(* CODESYS project Hylife_Repository

Project tree, tasks and I/O mapping:
  libraries: ; CXA_ModbusTCP, 1.8.0.3 (Bosch Rexroth AG)
  program PLC_PRG [ST]
*)

// PLC_PRG
PROGRAM PLC_PRG
VAR
	fbHandle_MB_CAN: FB_Handle_MB_CAN;
	//extra functie
	//Deze comment is toegevoegd vanuit een andere brench
	// test voor remote 2
	// test vor remote 
END_VAR

fbHandle_MB_CAN(I_MB_CAN:= MB_CAN_IO.I_MB_CAN);

END_PROGRAM
